FUNCTION F_ROUNDLREAL : LREAL
VAR_INPUT
	rValue		: LREAL; // Input Value
	iDecNumber	: INT; 	// Numbers after decimal point
END_VAR
VAR
	rOutValue	: LREAL;
	rLeftValue	: LREAL;
END_VAR

rOutValue := rValue * EXPT(10,iDecNumber);
rLeftValue := rOutValue - TRUNC(rOutValue);
IF rLeftValue >= 0.5 THEN
	rOutValue := TRUNC(rOutValue + 1) / EXPT(10,iDecNumber);
ELSE
	rOutValue := TRUNC(rOutValue) / EXPT(10,iDecNumber);
END_IF
F_ROUNDLREAL := rOutValue;

END_FUNCTION

(* stored: Version 1.1.0.1, ProductVersion 3.1.4024.9
   POU F_ROUNDLREAL: Id {625e7ba7-48bd-4cac-b9d8-1117997efc5b}, SpecialFunc None *)
